// TIA Portal project "Conveyor_Belt" (V18)

(* hardware
DEVICE "S7-1200 station_1"  S7-1200 Station
   slot 0: "Rack_0"  S7-1200 Rack  Rack  V1.0
   slot 1: "PLC_1"  CPU 1212C DC/DC/Rly  6ES7 212-1HE40-0XB0  V4.6
*)

// ===== PLC "PLC_1"  CPU 1212C DC/DC/Rly =====

VAR_GLOBAL   // PLC tag table "Default tag table"
   "start" AT %I0.0 : Bool;
   "stop" AT %I0.1 : Bool;
   "sensor1" AT %I0.2 : Bool;
   "sensor2" AT %I0.3 : Bool;
   "motor1" AT %Q0.0 : Bool;
   "motor2" AT %Q0.1 : Bool;
   "Tag_1" AT %M0.0 : Bool;
   "Tag_2" AT %MW0 : Int;
   "Tag_3" AT %M1.0 : Bool;
   "Tag_4" AT %MW1 : Int;
   "Tag_5" AT %M0.1 : Bool;
   "Tag_6" AT %M2.1 : Bool;
   "Tag_7" AT %M1.3 : Bool;
END_VAR

// folder: System blocks/Program resources

DATA_BLOCK "IEC_Counter_0_DB"   // DB1
{ S7_Optimized_Access := 'TRUE' }
AUTHOR : Simatic
FAMILY : IEC
NAME : CNTR
VERSION : 1.0
// stored: InstanceOfName IEC_COUNTER
"IEC_COUNTER"
BEGIN
END_DATA_BLOCK

DATA_BLOCK "IEC_Counter_0_DB_1"   // DB2
{ S7_Optimized_Access := 'TRUE' }
AUTHOR : Simatic
FAMILY : IEC
NAME : CNTR
VERSION : 1.0
// stored: InstanceOfName IEC_COUNTER
"IEC_COUNTER"
BEGIN
END_DATA_BLOCK

// folder: (top level)

ORGANIZATION_BLOCK "Main"   // OB1, LAD, ProgramCycle
TITLE = "Main Program Sweep (Cycle)"
{ S7_Optimized_Access := 'TRUE' }
VERSION : 0.1
   VAR_INPUT
      Initial_Call : Bool;   // Initial call of this OB
      Remanence : Bool;   // =True, if remanent data are available
   END_VAR
   VAR_TEMP   // added for the SCL form of the ladder/FBD networks
      _w1 : Bool;
   END_VAR
BEGIN

REGION Network 1
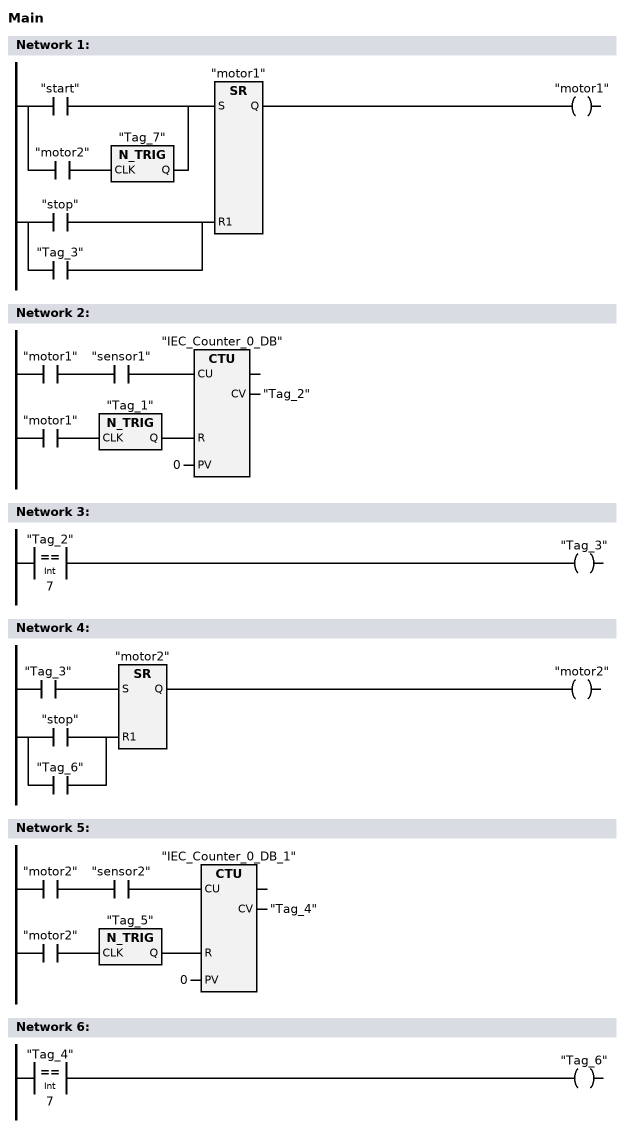
   RUNG wire#powerrail
      Contact( "start" )
      wire#w1
      S_SR(operand := "motor1", r1 := wire#w2)
      Coil( "motor1" )
   END_RUNG
   RUNG wire#powerrail
      Contact( "motor2" )
      N_Trig( "Tag_7" )
   END_RUNG wire#w1
   RUNG wire#powerrail
      Contact( "stop" )
   END_RUNG wire#w2
   RUNG wire#powerrail
      Contact( "Tag_3" )
   END_RUNG wire#w2
   // the same network as SCL:
   #_w1 := NOT "motor2" AND "Tag_7";   // falling edge
   "Tag_7" := "motor2";
   IF "start" OR #_w1 THEN
       "motor1" := TRUE;   // SR flip-flop
   END_IF;
   IF "stop" OR "Tag_3" THEN "motor1" := FALSE; END_IF;
   "motor1" := "motor1";
END_REGION

REGION Network 2
   #_w1 := NOT "motor1" AND "Tag_1";   // falling edge
   "Tag_1" := "motor1";
   "IEC_Counter_0_DB".CTU(CU := "motor1" AND "sensor1", R := #_w1, PV := 0, CV => "Tag_2");
END_REGION

REGION Network 3
   RUNG wire#powerrail
      { S7_Templates := "SrcType := Int" } EQ_Contact(in1 := "Tag_2", in2 := 7)
      Coil( "Tag_3" )
   END_RUNG
   // the same network as SCL:
   "Tag_3" := "Tag_2" = 7;
END_REGION

REGION Network 4
   RUNG wire#powerrail
      Contact( "Tag_3" )
      S_SR(operand := "motor2", r1 := wire#w1)
      Coil( "motor2" )
   END_RUNG
   RUNG wire#powerrail
      Contact( "stop" )
   END_RUNG wire#w1
   RUNG wire#powerrail
      Contact( "Tag_6" )
   END_RUNG wire#w1
   // the same network as SCL:
   IF "Tag_3" THEN
       "motor2" := TRUE;   // SR flip-flop
   END_IF;
   IF "stop" OR "Tag_6" THEN "motor2" := FALSE; END_IF;
   "motor2" := "motor2";
END_REGION

REGION Network 5
   #_w1 := NOT "motor2" AND "Tag_5";   // falling edge
   "Tag_5" := "motor2";
   "IEC_Counter_0_DB_1".CTU(CU := "motor2" AND "sensor2", R := #_w1, PV := 0, CV => "Tag_4");
END_REGION

REGION Network 6
   RUNG wire#powerrail
      { S7_Templates := "SrcType := Int" } EQ_Contact(in1 := "Tag_4", in2 := 7)
      Coil( "Tag_6" )
   END_RUNG
   // the same network as SCL:
   "Tag_6" := "Tag_4" = 7;
END_REGION
END_ORGANIZATION_BLOCK